// TIA Portal V18 export
DATA_BLOCK "AXES_Positions_Delays"   // DB33
{ S7_Optimized_Access := 'TRUE' }
VERSION : 0.1
// stored: AutoNumber true, DBAccessibleFromOPCUA true, IsOnlyStoredInLoadMemory false, IsRetainMemResEnabled false, IsWriteProtectedInAS false, MemoryReserve 100
   VAR
      AXIS_X_Position_DelayIn : Bool;
      AXIS_X_Position_DelayOut : Bool;
      AXIS_Y_Position_DelayIn : Bool;
      AXIS_Y_Position_DelayOut : Bool;
      AXIS_Z1_Position_DelayIn : Bool;
      AXIS_Z1_Position_DelayOut : Bool;
      AXIS_Z2_Position_DelayIn : Bool;
      AXIS_Z2_Position_DelayOut : Bool;
   END_VAR
BEGIN
END_DATA_BLOCK
